Omron CX-Programmer project NewProject (CX-Programmer 9.61)

# PLC NewPLC1: CP1E N30

## Global symbols (name address type ; comment)
0.00 BOOL  ; START_BUTTON
0.01 BOOL  ; STOP_BUTTON
100.00 BOOL  ; RELAY1
100.01 BOOL  ; RELAY2
100.02 BOOL  ; REALY3
100.03 BOOL  ; RELAY4
100.04 BOOL  ; RELAY5

## Program NewProgram1 (cyclic task 0)

### Section Main_Logic

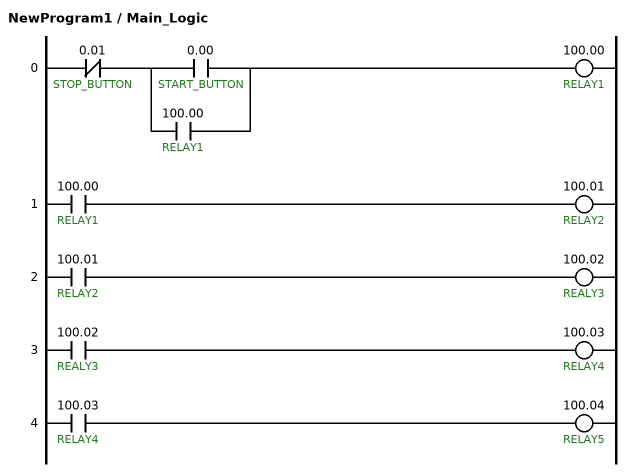
; rung 0
LDNOT 0.01  ; STOP_BUTTON
LD 0.00  ; START_BUTTON
OR 100.00  ; RELAY1
ANDLD
OUT 100.00  ; RELAY1
; rung 1
LD 100.00  ; RELAY1
OUT 100.01  ; RELAY2
; rung 2
LD 100.01  ; RELAY2
OUT 100.02  ; REALY3
; rung 3
LD 100.02  ; REALY3
OUT 100.03  ; RELAY4
; rung 4
LD 100.03  ; RELAY4
OUT 100.04  ; RELAY5
; rung 5
END(001)

### Section END
; rung 0
END(001)